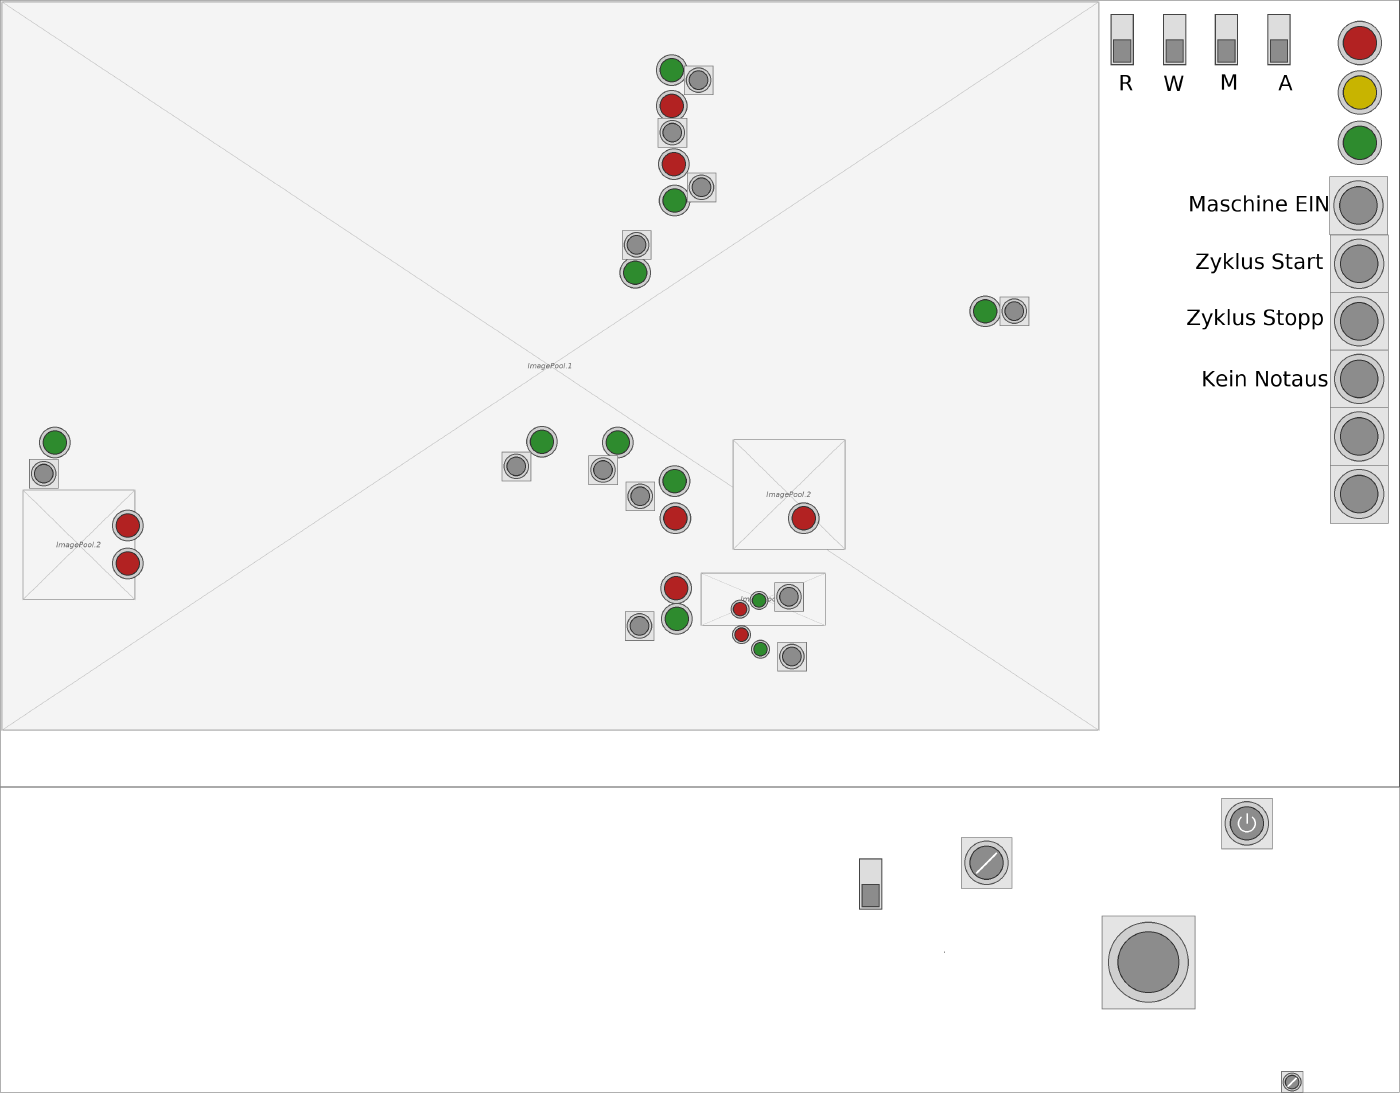
VISUALIZATION Visualization  // 1920x1500
    Rectangle (0,0 1920x1080)
    Image (2,2 1505x1000), image: ImagePool.1
    Image (1005,603 154x151), angle 26, image: ImagePool.2
    Image (31,672 154x151), image: ImagePool.2
    Lamp1 (1077,686 50x50), variable: MAIN.Saegeautomat.Ansteuerung_Ausgaenge.OUT_Saege_EIN, style: Lamp-Lamp1-Red
    Lamp1 (150,696 50x50), variable: MAIN.Saegeautomat.Ansteuerung_Ausgaenge.OUT_Zufuehrer_Antrieb_Vor, style: Lamp-Lamp1-Red
    Lamp1 (150,748 50x50), variable: MAIN.Saegeautomat.Ansteuerung_Ausgaenge.OUT_Zufuehrer_Antrieb_Rueck, style: Lamp-Lamp1-Red
    Lamp1 (1326,402 50x50), variable: MAIN.Saegeautomat.IN_Schaltausg_Lichtschranke, style: Lamp-Lamp1-Green
    Lamp1 (900,635 50x50), variable: MAIN.Saegeautomat.IN_Endl_Untere_Stammklemmung_Oben, style: Lamp-Lamp1-Green
    Lamp1 (903,824 50x50), variable: MAIN.Saegeautomat.IN_Endl_Untere_Stammklemmung_Unten, style: Lamp-Lamp1-Green
    Lamp1 (900,250 50x50), variable: MAIN.Saegeautomat.IN_Endl_Obere_Stammklemmung_Unten, style: Lamp-Lamp1-Green
    Lamp1 (896,71 50x50), variable: MAIN.Saegeautomat.IN_Endl_Obere_Stammklemmung_Oben, style: Lamp-Lamp1-Green
    Lamp1 (846,349 50x50), variable: MAIN.Saegeautomat.IN_Endl_Tastschiene, style: Lamp-Lamp1-Green
    Lamp1 (822,582 50x50), variable: MAIN.Saegeautomat.IN_Endl_Zufuehrer_Vorne, style: Lamp-Lamp1-Green
    Lamp1 (718,581 50x50), variable: MAIN.Saegeautomat.IN_Vorposition_Zufuehrer, style: Lamp-Lamp1-Green
    Lamp1 (50,582 50x50), variable: MAIN.Saegeautomat.IN_Endl_Zufuehrer_Hinten, style: Lamp-Lamp1-Green
    Image (961,786 171x72), angle 97, image: ImagePool.3
    Lamp1 (1028,876 30x30), variable: MAIN.Saegeautomat.IN_Endl_Saege_Oben, style: Lamp-Lamp1-Green
    Lamp1 (1026,809 30x30), variable: MAIN.Saegeautomat.IN_Endl_Saege_Unten, style: Lamp-Lamp1-Green
    Lamp1 (901,686 50x50), variable: MAIN.Saegeautomat.Ansteuerung_Ausgaenge.OUT_Stammklemmung_Unten_Hoch, style: Lamp-Lamp1-Red
    Lamp1 (902,782 50x50), variable: MAIN.Saegeautomat.Ansteuerung_Ausgaenge.OUT_Stammklemmung_Unten_Runter, style: Lamp-Lamp1-Red
    Lamp1 (899,200 50x50), variable: MAIN.Saegeautomat.Ansteuerung_Ausgaenge.OUT_Stammklemmung_Oben_Runter, style: Lamp-Lamp1-Red
    Lamp1 (896,120 50x50), variable: MAIN.Saegeautomat.Ansteuerung_Ausgaenge.OUT_Stammklemmung_Oben_Hoch, style: Lamp-Lamp1-Red
    Lamp1 (1000,821 30x30), variable: MAIN.Saegeautomat.Ansteuerung_Ausgaenge.OUT_Saege_Senken, style: Lamp-Lamp1-Red
    Lamp1 (1002,856 30x30), variable: MAIN.Saegeautomat.Ansteuerung_Ausgaenge.OUT_Saege_Heben, style: Lamp-Lamp1-Red
    RotarySwitch (1318,1149 70x70), behaviour: TOGGLE, style: Switch-RotarySwitch-Gray
    PushSwitch (1824,322 80x80), variable: MAIN.Saegeautomat.IN_Zyklus_Start, behaviour: TAP, style: Switch-PushSwitch-Gray
    PushSwitchLed (1293,1306 4x1), behaviour: TOGGLE, style: Switch-PushSwitchLed-Gray
    PushSwitchLed (1511,1254 128x133), behaviour: TOGGLE, style: Switch-PushSwitchLed-Gray
    DipSwitch (1159,1178 70x70), behaviour: TOGGLE, style: Switch-DipSwitch-Gray
    Lamp1 (1830,24 70x70), variable: MAIN.Saegeautomat.Steuerung_Meldeleuchten.OUT_Meldeleuchte_Rot, style: Lamp-Lamp1-Red
    Lamp1 (1830,92 70x70), variable: MAIN.Saegeautomat.Steuerung_Meldeleuchten.OUT_Meldeleuchte_Gelb, style: Lamp-Lamp1-Yellow
    Lamp1 (1830,161 70x70), variable: MAIN.Saegeautomat.Steuerung_Meldeleuchten.OUT_Meldeleuchte_Gruen, style: Lamp-Lamp1-Green
    PushSwitch (1824,401 80x80), variable: MAIN.Saegeautomat.IN_Zyklus_Stopp, behaviour: TAP, style: Switch-PushSwitch-Gray
    PushSwitch (1824,480 80x80), variable: MAIN.Saegeautomat.IN_Kein_Notaus, behaviour: TOGGLE, style: Switch-PushSwitch-Gray
    PushSwitch (1824,559 80x80), behaviour: TOGGLE, style: Switch-PushSwitch-Gray
    PushSwitch (1824,638 80x80), behaviour: TOGGLE, style: Switch-PushSwitch-Gray
    PushSwitch (1823,242 80x80), variable: MAIN.Saegeautomat.IN_Maschine_EIN, behaviour: TAP, style: Switch-PushSwitch-Gray
    PowerSwitch (1675,1095 70x70), behaviour: TOGGLE, style: Switch-PowerSwitch-Gray
    RotarySwitch (1697,1470 150x30), behaviour: TOGGLE, style: Switch-RotarySwitch-Gray
    DipSwitch (1719,19 70x70), variable: MAIN.Saegeautomat.IN_BetriebsArt_Automatik, behaviour: TOGGLE, style: Switch-DipSwitch-Gray
    DipSwitch (1647,19 70x70), variable: MAIN.Saegeautomat.IN_BetriebsArt_Manuell, behaviour: TOGGLE, style: Switch-DipSwitch-Gray
    DipSwitch (1504,19 70x70), variable: MAIN.Saegeautomat.IN_BetriebsArt_Referenz, behaviour: TOGGLE, style: Switch-DipSwitch-Gray
    DipSwitch (1576,19 70x70), variable: MAIN.Saegeautomat.IN_BetriebsArt_Warmlauf, behaviour: TOGGLE, style: Switch-DipSwitch-Gray
    Label (1583,344 235x30), "Zyklus Start"
    Label (1584,421 235x30), "Zyklus Stopp"
    Label (1590,505 235x30), "Kein Notaus"
    Label (1592,265 235x30), "Maschine EIN"
    Label (1517,99 40x30), "R"
    Label (1587,100 40x30), "W"
    Label (1661,98 40x30), "M"
    Label (1736,99 40x30), "A"
    PushSwitch (1062,799 40x40), variable: MAIN.Saegeautomat.IN_Endl_Saege_Unten, behaviour: TOGGLE, style: Switch-PushSwitch-Gray
    PushSwitch (1066,881 40x40), variable: MAIN.Saegeautomat.IN_Endl_Saege_Oben, behaviour: TOGGLE, style: Switch-PushSwitch-Gray
    PushSwitch (857,839 40x40), variable: MAIN.Saegeautomat.IN_Endl_Untere_Stammklemmung_Unten, behaviour: TOGGLE, style: Switch-PushSwitch-Gray
    PushSwitch (858,661 40x40), variable: MAIN.Saegeautomat.IN_Endl_Untere_Stammklemmung_Oben, behaviour: TOGGLE, style: Switch-PushSwitch-Gray
    PushSwitch (807,625 40x40), variable: MAIN.Saegeautomat.IN_Endl_Zufuehrer_Vorne, behaviour: TOGGLE, style: Switch-PushSwitch-Gray
    PushSwitch (688,620 40x40), variable: MAIN.Saegeautomat.IN_Vorposition_Zufuehrer, behaviour: TOGGLE, style: Switch-PushSwitch-Gray
    PushSwitch (40,630 40x40), variable: MAIN.Saegeautomat.IN_Endl_Zufuehrer_Hinten, behaviour: TOGGLE, style: Switch-PushSwitch-Gray
    PushSwitch (853,316 40x40), variable: MAIN.Saegeautomat.IN_Endl_Tastschiene, behaviour: TOGGLE, style: Switch-PushSwitch-Gray
    PushSwitch (942,237 40x40), variable: MAIN.Saegeautomat.IN_Endl_Obere_Stammklemmung_Unten, behaviour: TOGGLE, style: Switch-PushSwitch-Gray
    PushSwitch (938,90 40x40), variable: MAIN.Saegeautomat.IN_Endl_Obere_Stammklemmung_Oben, behaviour: TOGGLE, style: Switch-PushSwitch-Gray
    PushSwitch (1371,407 40x40), variable: MAIN.Saegeautomat.IN_Schaltausg_Lichtschranke, behaviour: TOGGLE, style: Switch-PushSwitch-Gray
    PushSwitch (902,162 40x40), variable: MAIN.Saegeautomat.IN_Schaltausg_Druckschalter_Obere_Klemmung, behaviour: TOGGLE, style: Switch-PushSwitch-Gray
END_VISUALIZATION

(* stored: Version 1.1.0.1, ProductVersion 3.1.4024.16
   Visu Visualization: Id {6a77ca1e-d980-421e-bbde-1ba80b5f5fe8} *)
